INTERFACE itfSynchronizedAxisCommand EXTENDS itfAxisCommand

PROPERTY InSync : BOOL
GET
END_GET
END_PROPERTY

END_INTERFACE

(* stored: Version 1.1.0.1, ProductVersion 3.1.4024.12
   Itf itfSynchronizedAxisCommand: Id {7dd525ce-dac1-4f6e-b84f-2915c80ad024}
   Property InSync: Id {1bd36755-586b-457f-9cff-65d3df788b01}
   Get Get: Id {2034d359-c895-42f9-bbe2-a343429f602f} *)
